{attribute 'qualified_only'}
VAR_GLOBAL
END_VAR

(* stored: Version 1.1.0.1, ProductVersion 3.1.4024.12
   GVL G_RealControlBox: Id {7355aca5-5201-4990-ae54-8098eeafaaf5} *)
